TYPE AxesDialogSign :
(
	DIALOG_PLUS := 0,
    DIALOG_MINUS := 1
);
END_TYPE

(* stored: Version 1.1.0.1, ProductVersion 3.1.4018.5
   DUT AxesDialogSign: Id {02feb5e7-c7c1-4507-bda5-725d72308f0b} *)
